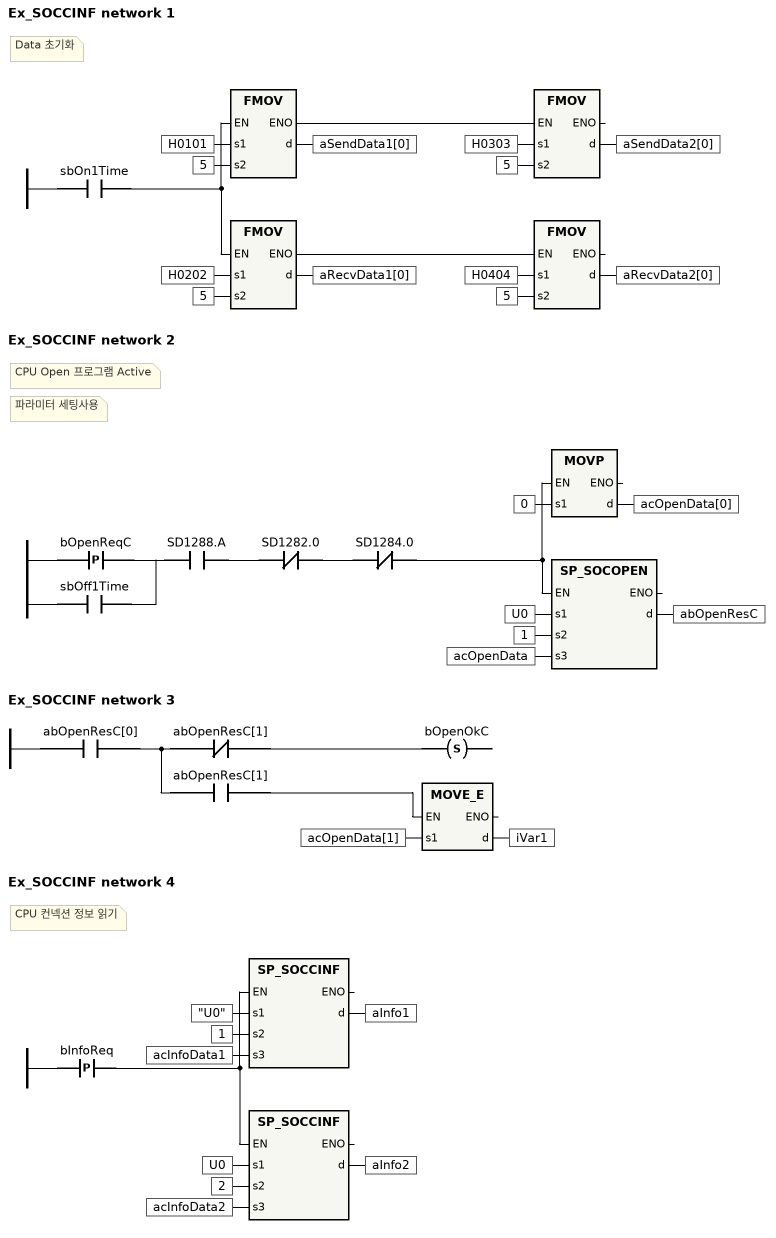
(* [picture p48: structured ladder/FBD of Ex_SOCCINF, networks 1 to 4] *)
(* network 1 *)
(* Data 초기화 *)
_e1 := FMOV(sbOn1Time, H0101, 5, aSendData1[0]);
FMOV(_e1, H0303, 5, aSendData2[0]);
_e2 := FMOV(sbOn1Time, H0202, 5, aRecvData1[0]);
FMOV(_e2, H0404, 5, aRecvData2[0]);
(* network 2 *)
(* CPU Open 프로그램 Active *)
(* 파라미터 세팅사용 *)
_p1 := (((LDP(TRUE, bOpenReqC) OR sbOff1Time) AND SD1288.A) AND NOT SD1282.0) AND NOT SD1284.0;
MOVP(_p1, 0, acOpenData[0]);
SP_SOCOPEN(_p1, U0, 1, acOpenData, abOpenResC);
(* network 3 *)
SET(abOpenResC[0] AND NOT abOpenResC[1], bOpenOkC);
MOVE_E(abOpenResC[0] AND abOpenResC[1], acOpenData[1], iVar1);
(* network 4 *)
(* CPU 컨넥션 정보 읽기 *)
_p1 := LDP(TRUE, bInfoReq);
SP_SOCCINF(_p1, "U0", 1, acInfoData1, aInfo1);
SP_SOCCINF(_p1, U0, 2, acInfoData2, aInfo2);
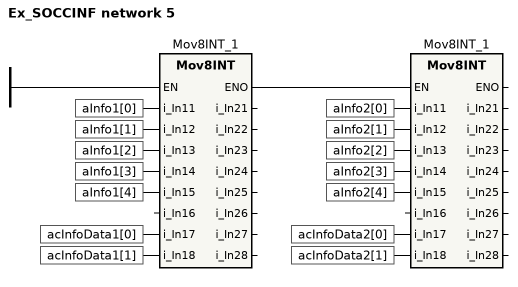
(* network 5 *)
Mov8INT_1(EN := TRUE, i_In11 := aInfo1[0], i_In12 := aInfo1[1], i_In13 := aInfo1[2], i_In14 := aInfo1[3], i_In15 := aInfo1[4], i_In17 := acInfoData1[0], i_In18 := acInfoData1[1]);
Mov8INT_1(EN := Mov8INT_1.ENO, i_In11 := aInfo2[0], i_In12 := aInfo2[1], i_In13 := aInfo2[2], i_In14 := aInfo2[3], i_In15 := aInfo2[4], i_In17 := acInfoData2[0], i_In18 := acInfoData2[1]);
END_PROGRAM

PROGRAM Ex_SLMPSND
VAR
  bSendReq : BOOL;
  Mov8WORD_1 : Mov8WORD;
  abSLMPRes : ARRAY [0..1] OF BOOL;
  acSLMPData : ARRAY [0..18] OF WORD;
  Mov8WORD_2 : Mov8WORD;
  Mov4WORD_1 : Mov4WORD;
  Mov8WORD_3 : Mov8WORD;
  Word2Bit16_1 : Word2Bit16;
  Word2Bit16_2 : Word2Bit16;
  Word2Bit16_3 : Word2Bit16;
  Word2Bit16_4 : Word2Bit16;
END_VAR
(* structured ladder/FBD written out as ST: instructions are called as NAME(EN, inputs, outputs); _pN, _eN, _tN stand for wires *)
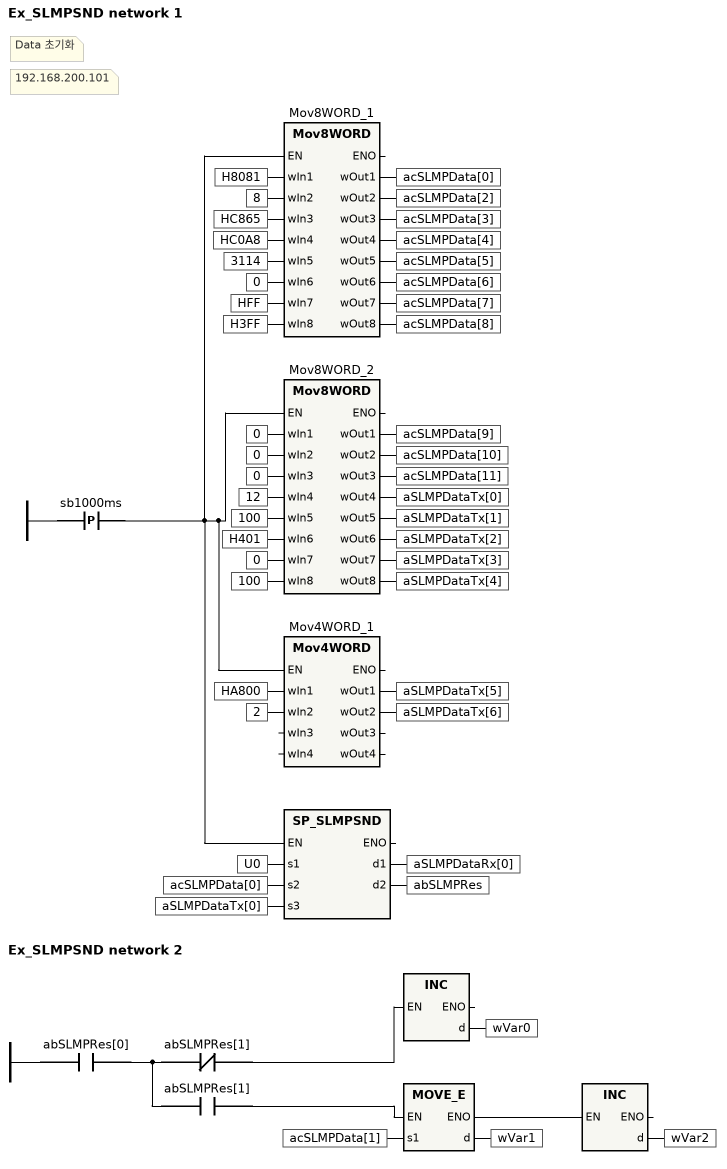
(* network 1 *)
(* Data 초기화 *)
(* 192.168.200.101 *)
_p1 := LDP(TRUE, sb1000ms);
Mov8WORD_1(EN := _p1, wIn1 := H8081, wIn2 := 8, wIn3 := HC865, wIn4 := HC0A8, wIn5 := 3114, wIn6 := 0, wIn7 := HFF, wIn8 := H3FF, wOut1 => acSLMPData[0], wOut2 => acSLMPData[2], wOut3 => acSLMPData[3], wOut4 => acSLMPData[4], wOut5 => acSLMPData[5], wOut6 => acSLMPData[6], wOut7 => acSLMPData[7], wOut8 => acSLMPData[8]);
Mov8WORD_2(EN := _p1, wIn1 := 0, wIn2 := 0, wIn3 := 0, wIn4 := 12, wIn5 := 100, wIn6 := H401, wIn7 := 0, wIn8 := 100, wOut1 => acSLMPData[9], wOut2 => acSLMPData[10], wOut3 => acSLMPData[11], wOut4 => aSLMPDataTx[0], wOut5 => aSLMPDataTx[1], wOut6 => aSLMPDataTx[2], wOut7 => aSLMPDataTx[3], wOut8 => aSLMPDataTx[4]);
Mov4WORD_1(EN := _p1, wIn1 := HA800, wIn2 := 2, wOut1 => aSLMPDataTx[5], wOut2 => aSLMPDataTx[6]);
SP_SLMPSND(_p1, U0, acSLMPData[0], aSLMPDataTx[0], aSLMPDataRx[0], abSLMPRes);
(* network 2 *)
INC(abSLMPRes[0] AND NOT abSLMPRes[1], wVar0);
_e1 := MOVE_E(abSLMPRes[0] AND abSLMPRes[1], acSLMPData[1], wVar1);
INC(_e1, wVar2);
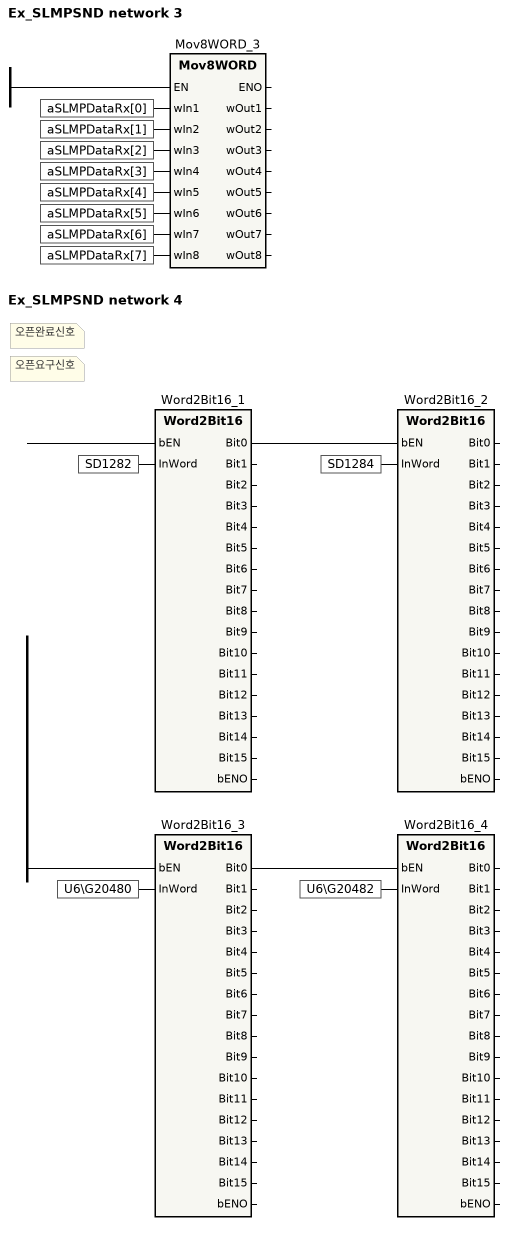
(* network 3 *)
Mov8WORD_3(EN := TRUE, wIn1 := aSLMPDataRx[0], wIn2 := aSLMPDataRx[1], wIn3 := aSLMPDataRx[2], wIn4 := aSLMPDataRx[3], wIn5 := aSLMPDataRx[4], wIn6 := aSLMPDataRx[5], wIn7 := aSLMPDataRx[6], wIn8 := aSLMPDataRx[7]);
(* network 4 *)
(* 오픈완료신호 *)
(* 오픈요구신호 *)
Word2Bit16_1(bEN := TRUE, InWord := SD1282);
Word2Bit16_2(bEN := Word2Bit16_1.Bit0, InWord := SD1284);
Word2Bit16_3(bEN := TRUE, InWord := U6\G20480);
Word2Bit16_4(bEN := Word2Bit16_3.Bit0, InWord := U6\G20482);
END_PROGRAM
